INTERFACE I_ChunkedRequestsManager

METHOD PUBLIC TryHandleIncomingRequest : BOOL
VAR_INPUT
	Request : I_Request;
	Response : I_ServerResponse;
	NextMidleware : I_Middleware;
END_VAR
END_METHOD

END_INTERFACE

(* stored: Version 1.1.0.1, ProductVersion 3.1.4024.12
   Itf I_ChunkedRequestsManager: Id {47686486-806a-45ce-8451-bf36c3eb2a47}
   Method TryHandleIncomingRequest: Id {6c30a40a-21ac-4901-9a48-7f2860d27987} *)
